# EPICS autosave request: ADApp/Db/NDROIN_settings.req
$(P)$(R)Use
$(P)$(R)ComputeStatistics
$(P)$(R)ComputeHistogram
$(P)$(R)BinX
$(P)$(R)BinY
$(P)$(R)MinX
$(P)$(R)MinY
$(P)$(R)SizeX
$(P)$(R)SizeY
$(P)$(R)ReverseX
$(P)$(R)ReverseY
$(P)$(R)HistSize
$(P)$(R)HistMin
$(P)$(R)HistMax
